FUNCTION_BLOCK E_DELAY (* Delayed event propagation *)
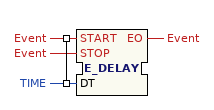
  EVENT_INPUT
    START WITH DT; (* Start delayed event propagation *)
    STOP; (* Stop the delayed event propagation *)
  END_EVENT
  EVENT_OUTPUT
    EO; (* Delayed event *)
  END_EVENT
  VAR_INPUT
    DT : TIME; (* Delay time, >0 *)
  END_VAR
  (* Service APPLICATION/RESOURCE: Delayed event propagation *)
END_FUNCTION_BLOCK
